// TIA Portal V20 export
TYPE "typeCmInterface"
// stored: Access Published, Namespace Unit1.Em5
   STRUCT
      softcam : "Unit1.Em5.typeCmInterfaceSoftCam";
      brakeTest : "Unit1.Em5.typeCmInterfaceBrakeTest";
   END_STRUCT;
END_TYPE
